{attribute addProperty BoxType "EJ2521-0224-0016"}
{attribute addProperty Id "PTO_StatusAT %I*PTO_Status_B9BB57FE1620ENC_Status_compactAT %I*ENC_Status_compact_FA080ECA4860PLS_Status_ChannelAT %I*ARRAY[0..1] OF PLS_Status_Channel_7A2392D13240PTO_ControlAT %Q*PTO_Control_0A6210C33240PTO_Target_compactAT %Q*PTO_Target_compact_C80C22BB1620ENC_Control_compactAT %Q*ENC_Control_compact_5C86AA9D3240PLS_Control_compact_ChannelAT %Q*ARRAY[0..1] OF PLS_Control_compact_Channel_F7E9C67496120WcStateAT %I*WcState_F855686C1620InfoDataAT %I*InfoData_BC63D37F80100"}
{attribute addProperty CRC "295026830"}
{attribute addProperty SizeInBites "368"}
{attribute addProperty SizeInBytes "46"}
TYPE EJ2521_F54ABF8F :
STRUCT
	{attribute addProperty Name "PTO_Status"}
	PTO_Status : PTO_Status_B9BB57FE;
	{attribute addProperty Name "ENC_Status_compact"}
	ENC_Status_compact : ENC_Status_compact_FA080ECA;
	{attribute addProperty Name "PLS_Status_Channel"}
	PLS_Status_Channel : ARRAY[0..1] OF PLS_Status_Channel_7A2392D1;
	{attribute addProperty Name "PTO_Control"}
	PTO_Control : PTO_Control_0A6210C3;
	{attribute addProperty Name "PTO_Target_compact"}
	PTO_Target_compact : PTO_Target_compact_C80C22BB;
	{attribute addProperty Name "ENC_Control_compact"}
	ENC_Control_compact : ENC_Control_compact_5C86AA9D;
	{attribute addProperty Name "PLS_Control_compact_Channel"}
	PLS_Control_compact_Channel : ARRAY[0..1] OF PLS_Control_compact_Channel_F7E9C674;
	{attribute addProperty Name "WcState"}
	WcState : WcState_F855686C;
	{attribute addProperty Name "InfoData"}
	InfoData : InfoData_BC63D37F;
END_STRUCT
END_TYPE

(* stored: Version 1.2.0.0, ProductVersion 3.1.4024.9
   DUT EJ2521_F54ABF8F: Id {056f7fda-7c8a-4808-935d-1fca40dc1629} *)
